RoboDK station: Arctos pick and place.rdk

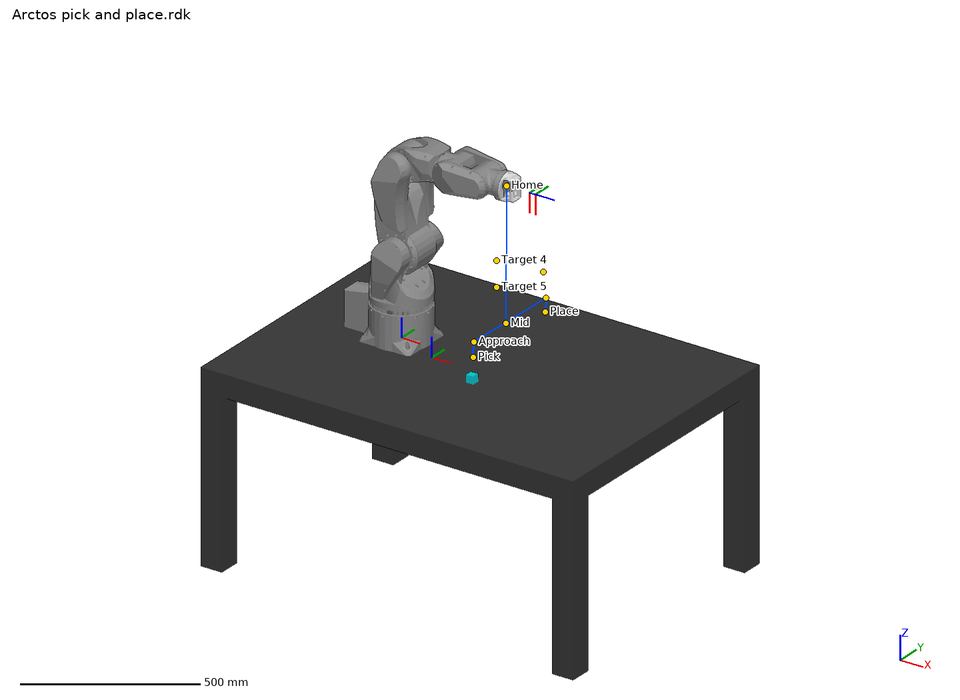
[picture v0: the station drawn from its stored meshes, robots at their saved joint values, targets as dots, program paths as lines]
Station Arctos pick and place (saved by RoboDK 5.6.8). Poses are relative to the parent item; angles as X-Y-Z fixed-axis rotations.
  - object b at (0, 0, 0) mm, size 269.1 x 183.6 x 136 mm, geometry from b.step
  - object J1 at (0, 0, 0) mm, size 183.8 x 217.5 x 313.9 mm, geometry from J1.step
  - object J2 (1) at (0, 0, 0) mm, size 144.2 x 196.7 x 374.9 mm, geometry from J2 (1).step
  - object J3 at (0, 0, 0) mm, size 176.8 x 123.2 x 122.2 mm, geometry from J3.step
  - object J4 (1) at (0, 0, 0) mm, size 217.1 x 158.5 x 97.3 mm, geometry from J4 (1).step
  - object J5 at (0, 0, 0) mm, size 118.7 x 78.5 x 80.7 mm, geometry from J5.step
  - object J6 (1) at (0, 0, 0) mm, size 18.5 x 86 x 86 mm, geometry from J6 (1).step
  - frame My Mechanism Base at (899.78, 999.44, 57.25) mm
    - robot Arctos: 6 axes
        modified DH rows (alpha deg, a mm, theta deg, d mm): 0, 0, 0, 287.872; -90, 20.174, -90, 0; 0, 260.986, 0, 0; -90, 19.219, 0, 260.753; 90, 0, 0, 0; -90, 0, 180, 74.745
        joint limits [-200, -125, -50, -200, -100, -200] to [200, 75, 100, 200, 100, 200]; home [0, 0, 0, 0, 0, 0]; saved at [0, 0, 0, 0, 0, 0]
      - frame gv1 Base at (0.55, 2.41, 96.13) mm
        - robot gv1: 1 axes
            joint limits [0] to [29]; home [0]; saved at [29]
        - target Open (joint target) at (0, 0, 150) mm; joints [29, -11.232, -27.921, 0, -39.154, 0] of gv1
        - target Close (joint target) at (0, 0, 150) mm; joints [0, -11.232, -27.921, 0, -39.154, 0] of gv1
        - frame Frame 4 at (0, 0, -20) mm
      - tool Tool 1, TCP at (0, 0, 0) mm
    - target Home (Cartesian target) at (355.67, 0, 568.08) mm, rotated rx 0 ry 90 rz 0 deg; joints [0, 0, 0, 0, 0, 0] of Arctos
    - target Target 4 (Cartesian target) at (321.25, 0, 328.47) mm, rotated rx -180 ry 1.24 rz 180 deg; joints [0, -16.767, -18.424, 0, 53.569, 0] of Arctos
    - target Target 5 (Cartesian target) at (323.05, 0, 245.49) mm, rotated rx -180 ry 1.24 rz 180 deg; joints [0, -29.246, -23.322, 0, 36.192, 0] of Arctos
    - target Target 6 (joint target) at (327.83, 2.41, -0.6) mm, rotated rx 180 ry 1.24 rz -180 deg; joints [29] of gv1
    - target Target 7 (Cartesian target) at (355.67, 0, 568.08) mm, rotated rx 0 ry 90 rz 0 deg; joints [0, 0, 0, 0, 0, 0] of Arctos
    - target Target 8 (Cartesian target) at (323.92, 223.71, 205.45) mm, rotated rx -180 ry 1.24 rz 180 deg; joints [34.765, -46.57, -3.34, 1.121, 39.077, 35.629] of Arctos
    - frame Frame 3 at (200, -140.56, 51.54) mm
    - object X upper Core_1-X upper core-stl at (350, 30, -160) mm, size 183.7 x 183.6 x 54 mm, geometry from X upper Core_1-X upper core-stl.stl
    - object arctos table v1 at (-350, 430, -40) mm, rotated rx 90 ry 0 rz 0 deg, size 1260 x 612 x 900 mm, geometry from arctos table v1.step
    - target Approach (Cartesian target) at (325.78, -115.96, 125.08) mm, rotated rx -180 ry -2.12 rz 180 deg; joints [-19.441, -55.543, -13.057, 1.774, 23.408, -17.8] of Arctos
    - target Pick (Cartesian target) at (324, -115.96, 76.82) mm, rotated rx -180 ry -2.12 rz 180 deg; joints [-19.539, -65.245, -8.942, 2.315, 17.824, -17.323] of Arctos
    - target App place (Cartesian target) at (325.64, 233.79, 121.21) mm, rotated rx -180 ry -2.12 rz -180 deg; joints [35.448, -62.381, 3.631, -2.256, 32.995, 33.537] of Arctos
    - target Place (Cartesian target) at (324, 233.79, 76.82) mm, rotated rx 180 ry -2.12 rz -180 deg; joints [35.583, -70.486, 7.514, -2.561, 28.776, 33.32] of Arctos
    - target Mid (Cartesian target) at (325.64, 39.03, 121.21) mm, rotated rx 180 ry -2.12 rz -180 deg; joints [6.778, -54.74, -17.596, -0.739, 19.769, 6.078] of Arctos
  - object Left jaw-step at (0, 0, -26) mm, size 32.5 x 34 x 45.7 mm, geometry from Left jaw-step.stp
  - object Right jaw-step at (-15, 0, -26) mm, size 32.5 x 31.3 x 45.7 mm, geometry from Right jaw-step.stp
  - object Gripper carriage-step at (0, 0, 0) mm, size 85.7 x 85.9 x 35.9 mm, geometry from Gripper carriage-step.stp
  - program Open (3 instructions, listed below)
  - program Close (3 instructions, listed below)
  - program Prog3 (15 instructions, listed below)
  - object box v0 at (1231.57, 871.43, 82.22) mm, rotated rx 180 ry 2.12 rz -180 deg, size 25 x 25 x 25 mm, geometry from box v0.step
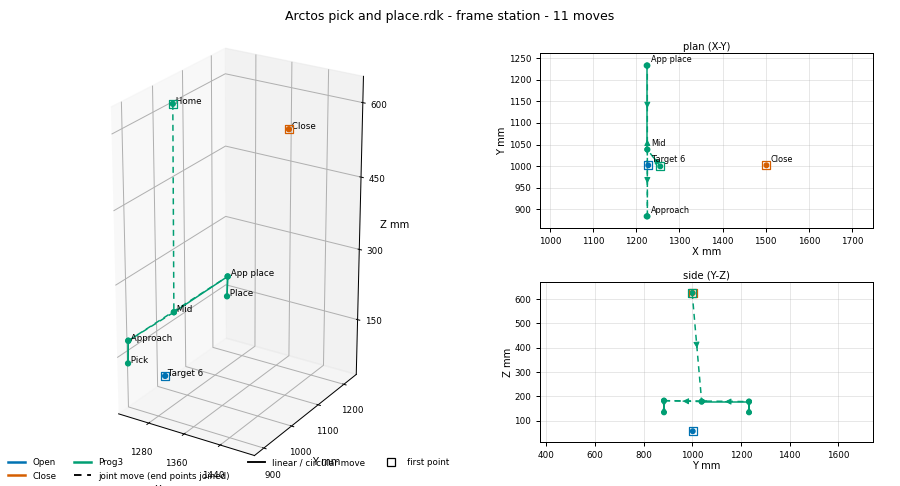
[picture p0: tool path of Arctos pick and place.rdk in frame station, 11 of 11 moves have a stored position in this frame; points joined in program order, loops and branches not executed]

--- program Open (robot gv1) ---
  Set Ref.: gv1 Base
  Set Tool: Tool at (0, 0, 0) mm
  MoveJ (Target 6)

--- program Close (robot gv1) ---
  Set Ref.: gv1 Base
  Set Tool: Tool at (0, 0, 0) mm
  MoveJ (Close)

--- program Prog3 (robot Arctos) ---
  Set Ref.: My Mechanism Base
  Set Tool: Tool 1
  MoveJ (Home)
  MoveJ (Mid)
  MoveJ (Approach)
  MoveL (Pick)
  Call Close
  Attach to Tool 1
  MoveL (Approach)
  MoveJ (App place)
  MoveL (Place)
  Call Open
  Detach from Tool 1
  MoveL (App place)
  MoveL (Mid)
